FUNCTION alg_g_algeb1: REAL
{ S7_Optimized_Access := 'false' }
    VAR_INPUT
        state: STATE;
    END_VAR

BEGIN
    alg_g_algeb1 := (state.curTime) + (1.0);
END_FUNCTION
